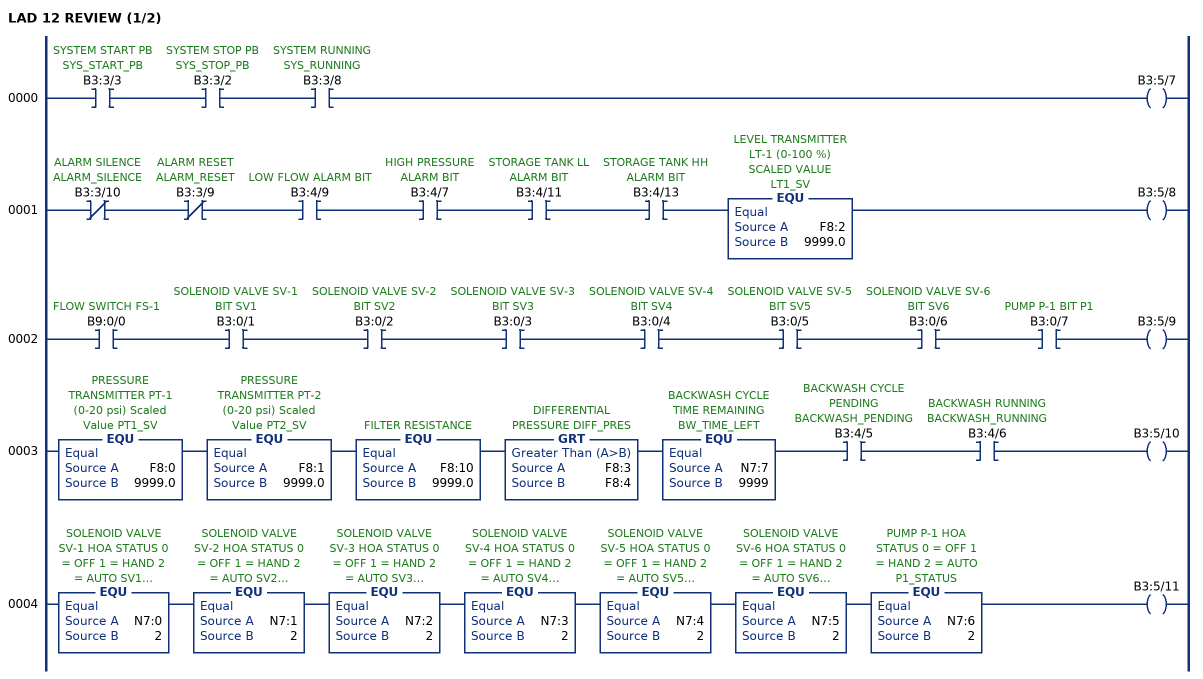
% Rung: 0 %
SOR XIC B3:3/3 XIC B3:3/2 XIC B3:3/8 OTE B3:5/7 EOR
%   B3:3/3  SYS_START_PB  "SYSTEM START PB" %
%   B3:3/2  SYS_STOP_PB  "SYSTEM STOP PB" %
%   B3:3/8  SYS_RUNNING  "SYSTEM RUNNING" %
% Rung: 1 %
SOR XIO B3:3/10 XIO B3:3/9 XIC B3:4/9 XIC B3:4/7 XIC B3:4/11 XIC B3:4/13 EQU F8:2 9999.0 OTE B3:5/8 EOR
%   B3:3/10  ALARM_SILENCE  "ALARM SILENCE" %
%   B3:3/9  ALARM_RESET  "ALARM RESET" %
%   B3:4/9  "LOW FLOW ALARM BIT" %
%   B3:4/7  "HIGH PRESSURE ALARM BIT" %
%   B3:4/11  "STORAGE TANK LL ALARM BIT" %
%   B3:4/13  "STORAGE TANK HH ALARM BIT" %
%   F8:2  LT1_SV  "LEVEL TRANSMITTER LT-1 (0-100 %) SCALED VALUE" %
% Rung: 2 %
SOR XIC B9:0/0 XIC B3:0/1 XIC B3:0/2 XIC B3:0/3 XIC B3:0/4 XIC B3:0/5 XIC B3:0/6 XIC B3:0/7 OTE B3:5/9 EOR
%   B9:0/0  "FLOW SWITCH FS-1" %
%   B3:0/1  SV1  "SOLENOID VALVE SV-1 BIT" %
%   B3:0/2  SV2  "SOLENOID VALVE SV-2 BIT" %
%   B3:0/3  SV3  "SOLENOID VALVE SV-3 BIT" %
%   B3:0/4  SV4  "SOLENOID VALVE SV-4 BIT" %
%   B3:0/5  SV5  "SOLENOID VALVE SV-5 BIT" %
%   B3:0/6  SV6  "SOLENOID VALVE SV-6 BIT" %
%   B3:0/7  P1  "PUMP P-1 BIT" %
% Rung: 3 %
SOR EQU F8:0 9999.0 EQU F8:1 9999.0 EQU F8:10 9999.0 GRT F8:3 F8:4 EQU N7:7 9999 XIC B3:4/5 XIC B3:4/6 OTE B3:5/10 EOR
%   F8:0  PT1_SV  "PRESSURE TRANSMITTER PT-1 (0-20 psi) Scaled Value" %
%   F8:1  PT2_SV  "PRESSURE TRANSMITTER PT-2 (0-20 psi) Scaled Value" %
%   F8:10  "FILTER RESISTANCE" %
%   F8:3  DIFF_PRES  "DIFFERENTIAL PRESSURE" %
%   F8:4  BACKWASH_SP  "Backwash Cycle Trigger Setpoint" %
%   N7:7  BW_TIME_LEFT  "BACKWASH CYCLE TIME REMAINING" %
%   B3:4/5  BACKWASH_PENDING  "BACKWASH CYCLE PENDING" %
%   B3:4/6  BACKWASH_RUNNING  "BACKWASH RUNNING" %
% Rung: 4 %
SOR EQU N7:0 2 EQU N7:1 2 EQU N7:2 2 EQU N7:3 2 EQU N7:4 2 EQU N7:5 2 EQU N7:6 2 OTE B3:5/11 EOR
%   N7:0  SV1_STATUS  "SOLENOID VALVE SV-1 HOA STATUS 0 = OFF 1 = HAND 2 = AUTO" %
%   N7:1  SV2_STATUS  "SOLENOID VALVE SV-2 HOA STATUS 0 = OFF 1 = HAND 2 = AUTO" %
%   N7:2  SV3_STATUS  "SOLENOID VALVE SV-3 HOA STATUS 0 = OFF 1 = HAND 2 = AUTO" %
%   N7:3  SV4_STATUS  "SOLENOID VALVE SV-4 HOA STATUS 0 = OFF 1 = HAND 2 = AUTO" %
%   N7:4  SV5_STATUS  "SOLENOID VALVE SV-5 HOA STATUS 0 = OFF 1 = HAND 2 = AUTO" %
%   N7:5  SV6_STATUS  "SOLENOID VALVE SV-6 HOA STATUS 0 = OFF 1 = HAND 2 = AUTO" %
%   N7:6  P1_STATUS  "PUMP P-1 HOA STATUS 0 = OFF 1 = HAND 2 = AUTO" %

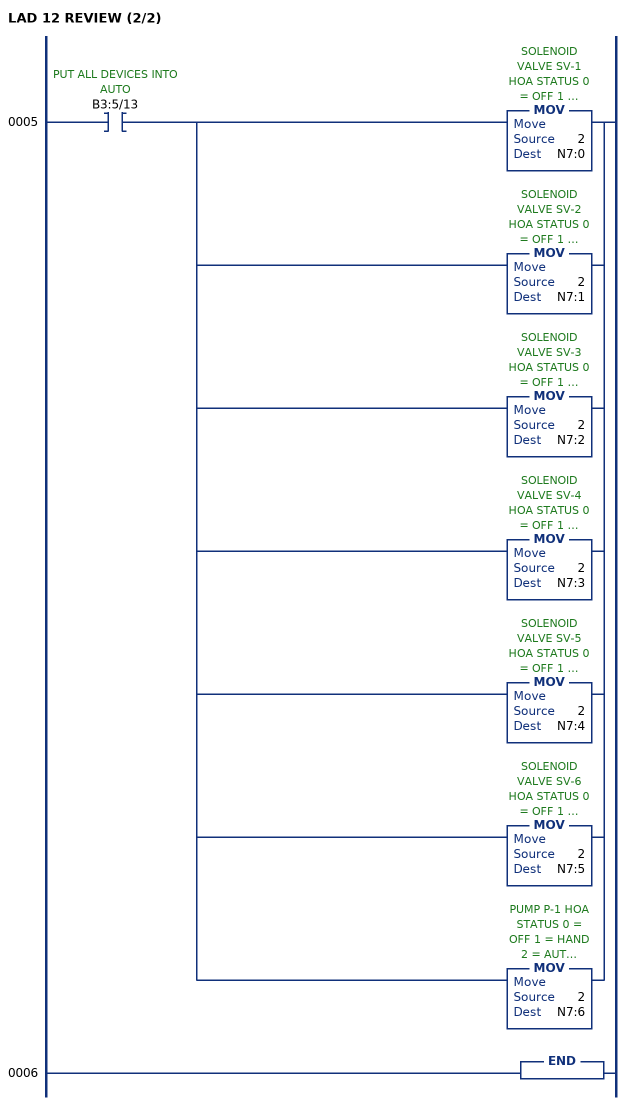
% Rung: 5 %
SOR XIC B3:5/13 BST MOV 2 N7:0 NXB MOV 2 N7:1 NXB MOV 2 N7:2 NXB MOV 2 N7:3 NXB MOV 2 N7:4 NXB MOV 2 N7:5 NXB MOV 2 N7:6 BND EOR
%   B3:5/13  "PUT ALL DEVICES INTO AUTO" %
%   N7:0  SV1_STATUS  "SOLENOID VALVE SV-1 HOA STATUS 0 = OFF 1 = HAND 2 = AUTO" %
%   N7:1  SV2_STATUS  "SOLENOID VALVE SV-2 HOA STATUS 0 = OFF 1 = HAND 2 = AUTO" %
%   N7:2  SV3_STATUS  "SOLENOID VALVE SV-3 HOA STATUS 0 = OFF 1 = HAND 2 = AUTO" %
%   N7:3  SV4_STATUS  "SOLENOID VALVE SV-4 HOA STATUS 0 = OFF 1 = HAND 2 = AUTO" %
%   N7:4  SV5_STATUS  "SOLENOID VALVE SV-5 HOA STATUS 0 = OFF 1 = HAND 2 = AUTO" %
%   N7:5  SV6_STATUS  "SOLENOID VALVE SV-6 HOA STATUS 0 = OFF 1 = HAND 2 = AUTO" %
%   N7:6  P1_STATUS  "PUMP P-1 HOA STATUS 0 = OFF 1 = HAND 2 = AUTO" %
% Rung: 6 %
SOR END EOR

OTHER DOCUMENTED ADDRESSES
  DFILE:0  "OUTPUT"
  DFILE:1  "INPUT"
  DFILE:2  "STATUS"
  DFILE:3  "BINARY"
  DFILE:4  "TIMER"
  DFILE:5  "COUNTER"
  DFILE:6  "CONTROL"
  DFILE:7  "INTEGER"
  DFILE:8  "FLOAT"
  DFILE:9  "DIGITAL IO"
  DFILE:10  "ANALOG IO"

DATA TABLE (non-zero values as saved)
DATA B3
% B3:0 % 0X0000 0X0000 0X0000 0X0028 0X1802 0X0000 0X0020
DATA T4
% .PRE .ACC %
% T4:0 % 5 0
% T4:1 % 5 0
% T4:2 % 5 0
% T4:3 % 5 5
% T4:4 % 5 0
% T4:5 % 2 0
% T4:6 % 60 0
% T4:7 % 2 0
% T4:8 % 2 0
% T4:9 % 500 500
% T4:10 % 2 0
% T4:11 % 5 0
% T4:12 % 500 0
% T4:13 % 60 0
% T4:14 % 5 0
DATA N7
% N7:0 % 0 0 0 0 0 0 0 60 0 0
DATA F8
% F8:0 % 0 0 0 0 5
% F8:5 % 15 10 90 20 80
% F8:10 % 400 0
